// TIA Portal V19 export
TYPE "lexchangetray_typeUnEmn_toRollerReq"
// Type: Bool
// stored: Access Published
   STRUCT
      outFeedReq : Bool;   // Manual mode parameters for axis control interface
   END_STRUCT;
END_TYPE
